{attribute addProperty BoxType "EK1100-0000-0018"}
{attribute addProperty Id "Beckhoff_EKM1xxxEK1122Beckhoff_EKM1xxxEK1122_D80A806C2901362.625"}
{attribute addProperty CRC "1116840916"}
{attribute addProperty SizeInBites "2901"}
{attribute addProperty SizeInBytes "362.625"}
TYPE Beckhoff_EKM1xxx_4291A3D4 EXTENDS EK1100_179A0949 :
STRUCT
	{attribute addProperty Name "Beckhoff_EKM1xxxEK1122"}
	Beckhoff_EKM1xxxEK1122 : Beckhoff_EKM1xxxEK1122_D80A806C;
END_STRUCT
END_TYPE

(* stored: Version 1.2.0.0, ProductVersion 3.1.4024.9
   DUT Beckhoff_EKM1xxx_4291A3D4: Id {8f7b1cb8-ca6a-4709-a62e-a16069e9ff15} *)
